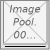
VISUALIZATION F_MainMenu_00  // 50x50
VAR_IN_OUT
	stMenuButton	: ST_HMIEButton_HMI;
END_VAR
    Image (3,0 44x44), invisible if: not stMenuButton.bVisible, image: ImagePool.00_MainScreen
        OnMouseDown: execute { stMenuButton.bPushed := TRUE; }
    Line (5,46) (45,46), invisible if: not stMenuButton.bVisible or not stMenuButton.bActive, input disabled if: not stMenuButton.bEnable
END_VISUALIZATION

(* stored: Version 1.1.0.1
   Visu F_MainMenu_00: Id {e74dab01-5e5b-4bb2-9173-728c4ab59589} *)
